KUKA KRL program: wkz4_off_st600.src, wkz4_off_st600.dat

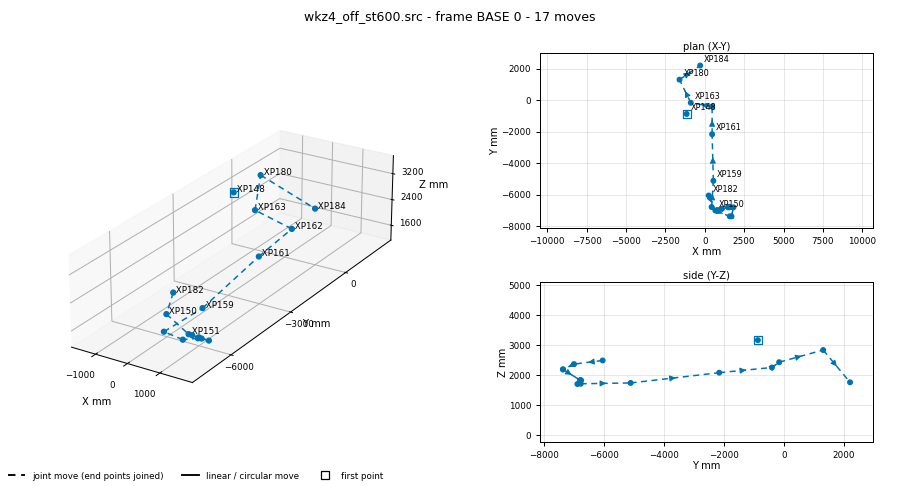
[picture p0: tool path of wkz4_off_st600.src in frame BASE 0, 17 of 18 moves have a stored position in this frame; points joined in program order, loops and branches not executed]
--- wkz4_off_st600.src ---
&ACCESS RVO1
&REL 256
&COMMENT Pega Griper ACCELO Geobox
&PARAM DISKPATH = KRC:\R1\Program
DEF wkz4_off_st600( )
;FOLD INI
  ;FOLD BASISTECH INI
    GLOBAL INTERRUPT DECL 3 WHEN $STOPMESS==TRUE DO IR_STOPM ( )
    INTERRUPT ON 3
    BAS (#INITMOV,0 )
  ;ENDFOLD (BASISTECH INI)
;FOLD GRIPPERTECH INI
USER_GRP(0,DUMMY,DUMMY,GDEFAULT)
;ENDFOLD (GRIPPERTECH INI)
  ;FOLD USER INI
    ;Make your modifications here

  ;ENDFOLD (USER INI)
;ENDFOLD (INI)

; Caracterização dos meios de produção:
; Versão Atual:
; 12/07/2013 12:00 Name: P13.050-R3 CHANGES: Pega Gripper na Geo
; Accelo

chk_w8_wechs_ok ( )       ; CHECK TOOLCHANGER

;FOLD PTP P148 CONT Vel=100 % PDAT114 Tool[4]:Gripper Lateral E.Accelo Base[0];%{PE}%R 8.2.20,%MKUKATPBASIS,%CMOVE,%VPTP,%P 1:PTP, 2:P148, 3:C_DIS, 5:100, 7:PDAT114
$BWDSTART=FALSE
PDAT_ACT=PPDAT114
FDAT_ACT=FP148
BAS(#PTP_PARAMS,100)
PTP XP148 C_DIS
;ENDFOLD
;FOLD PTP P172 CONT Vel=100 % PDAT131 Tool[4]:Gripper Lateral E.Accelo Base[0];%{PE}%R 8.2.20,%MKUKATPBASIS,%CMOVE,%VPTP,%P 1:PTP, 2:P172, 3:C_DIS, 5:100, 7:PDAT131
$BWDSTART=FALSE
PDAT_ACT=PPDAT131
FDAT_ACT=FP172
BAS(#PTP_PARAMS,100)
PTP XP172 C_DIS
;ENDFOLD
;FOLD PTP P182 Vel=100 % PDAT143 Tool[8]:Tool Changer Base[0];%{PE}%R 8.2.20,%MKUKATPBASIS,%CMOVE,%VPTP,%P 1:PTP, 2:P182, 3:, 5:100, 7:PDAT143
$BWDSTART=FALSE
PDAT_ACT=PPDAT143
FDAT_ACT=FP182
BAS(#PTP_PARAMS,100)
PTP XP182
;ENDFOLD


;FOLD OUT 3337 'R3 retira garra Geo' State=TRUE ;%{PE}%R 8.2.20,%MKUKATPBASIS,%COUT,%VOUTX,%P 2:3337, 3:R3 retira garra Geo, 5:TRUE, 6:
$OUT[3337]=TRUE
;ENDFOLD
;FOLD WAIT FOR ( IN 3337 'Aguarda Lib. entrar Geo' );%{PE}%R 8.2.20,%MKUKATPBASIS,%CEXT_WAIT_FOR,%VEXT_WAIT_FOR,%P 2:, 4:, 5:$IN, 6:3337, 7:Aguarda Lib. entrar Geo, 9:
WAIT FOR  ( $IN[3337] )
;ENDFOLD
;FOLD OUT 3337 'R3 retira garra Geo' State=FALSE ;%{PE}%R 8.2.20,%MKUKATPBASIS,%COUT,%VOUTX,%P 2:3337, 3:R3 retira garra Geo, 5:FALSE, 6:
$OUT[3337]=FALSE
;ENDFOLD
;FOLD OUT 3348 'Fora area GEOBOX' State=FALSE ;%{PE}%R 8.2.20,%MKUKATPBASIS,%COUT,%VOUTX,%P 2:3348, 3:Fora area GEOBOX, 5:FALSE, 6:
$OUT[3348]=FALSE
;ENDFOLD

;FOLD Collision.Monitoring_AREA_3_On ;%{PE}%MKUKATPUSER
COLLSTOP( 9, 1 ) ;not Interrupt-Controlled
;ENDFOLD
;FOLD Collision.Monitoring_AREA_5_On ;%{PE}%MKUKATPUSER
COLLSTOP( 11, 1 ) ;not Interrupt-Controlled
;ENDFOLD

;FOLD PTP P150 CONT Vel=100 % PDAT116 Tool[4]:Gripper Lateral E.Accelo Base[0];%{PE}%R 8.2.20,%MKUKATPBASIS,%CMOVE,%VPTP,%P 1:PTP, 2:P150, 3:C_DIS, 5:100, 7:PDAT116
$BWDSTART=FALSE
PDAT_ACT=PPDAT116
FDAT_ACT=FP150
BAS(#PTP_PARAMS,100)
PTP XP150 C_DIS
;ENDFOLD
;FOLD PTP P151 CONT Vel=100 % PDAT117 Tool[4]:Gripper Lateral E.Accelo Base[0];%{PE}%R 8.2.20,%MKUKATPBASIS,%CMOVE,%VPTP,%P 1:PTP, 2:P151, 3:C_DIS, 5:100, 7:PDAT117
$BWDSTART=FALSE
PDAT_ACT=PPDAT117
FDAT_ACT=FP151
BAS(#PTP_PARAMS,100)
PTP XP151 C_DIS
;ENDFOLD

;FOLD OUT 224 'Bloquear MPS' State=FALSE ;%{PE}%R 8.2.20,%MKUKATPBASIS,%COUT,%VOUTX,%P 2:224, 3:Bloquear MPS, 5:FALSE, 6:
$OUT[224]=FALSE
;ENDFOLD
;FOLD OUT 223 'Desbloquear MPS' State=TRUE ;%{PE}%R 8.2.20,%MKUKATPBASIS,%COUT,%VOUTX,%P 2:223, 3:Desbloquear MPS, 5:TRUE, 6:
$OUT[223]=TRUE
;ENDFOLD
;FOLD WAIT FOR ( IN 217 'MPS Destravado' );%{PE}%R 8.2.20,%MKUKATPBASIS,%CEXT_WAIT_FOR,%VEXT_WAIT_FOR,%P 2:, 4:, 5:$IN, 6:217, 7:MPS Destravado, 9:
WAIT FOR  ( $IN[217] )
;ENDFOLD
;FOLD WAIT FOR NOT ( IN 221 'MPS Travado' );%{PE}%R 8.2.20,%MKUKATPBASIS,%CEXT_WAIT_FOR,%VEXT_WAIT_FOR,%P 2:NOT, 4:, 5:$IN, 6:221, 7:MPS Travado, 9:
WAIT FOR  NOT ( $IN[221] )
;ENDFOLD

;FOLD ; PONTO DE PEGA DO GRIPPER;%{PE}%R 5.4.33,%MKUKATPBASIS,%CCOMMENT,%VNORMAL,%P 2:PONTO DE PEGA DO GRIPPER
;ENDFOLD
;FOLD LIN P179 Vel=2 m/s CPDAT55 Tool[8]:Tool Changer Base[0];%{PE}%R 8.2.20,%MKUKATPBASIS,%CMOVE,%VLIN,%P 1:LIN, 2:P179, 3:, 5:2, 7:CPDAT55
$BWDSTART=FALSE
LDAT_ACT=LCPDAT55
FDAT_ACT=FP179
BAS(#CP_PARAMS,2)
LIN XP179
;ENDFOLD

;FOLD WAIT Time=0.5 sec;%{PE}%R 8.2.20,%MKUKATPBASIS,%CWAIT,%VWAIT,%P 3:0.5
WAIT SEC 0.5
;ENDFOLD
;FOLD WAIT FOR ( IN 219 'Posicao p/ Acoplamento OK' );%{PE}%R 8.2.20,%MKUKATPBASIS,%CEXT_WAIT_FOR,%VEXT_WAIT_FOR,%P 2:, 4:, 5:$IN, 6:219, 7:Posicao p/ Acoplamento OK, 9:
WAIT FOR  ( $IN[219] )
;ENDFOLD
;FOLD OUT 223 'Desbloquear MPS' State=FALSE ;%{PE}%R 8.2.20,%MKUKATPBASIS,%COUT,%VOUTX,%P 2:223, 3:Desbloquear MPS, 5:FALSE, 6:
$OUT[223]=FALSE
;ENDFOLD
;FOLD OUT 224 'Bloquear MPS' State=TRUE ;%{PE}%R 8.2.20,%MKUKATPBASIS,%COUT,%VOUTX,%P 2:224, 3:Bloquear MPS, 5:TRUE, 6:
$OUT[224]=TRUE
;ENDFOLD
;FOLD WAIT FOR NOT ( IN 217 'MPS Destravado' );%{PE}%R 8.2.20,%MKUKATPBASIS,%CEXT_WAIT_FOR,%VEXT_WAIT_FOR,%P 2:NOT, 4:, 5:$IN, 6:217, 7:MPS Destravado, 9:
WAIT FOR  NOT ( $IN[217] )
;ENDFOLD
;FOLD WAIT FOR ( IN 221 'MPS Travado' );%{PE}%R 8.2.20,%MKUKATPBASIS,%CEXT_WAIT_FOR,%VEXT_WAIT_FOR,%P 2:, 4:, 5:$IN, 6:221, 7:MPS Travado, 9:
WAIT FOR  ( $IN[221] )
;ENDFOLD
;FOLD IBUS ON SEGMENT_3;%{PE}%R 8.2.20,%MKUKATPBASIS,%CIBUS,%VMAP,%P 2:#ON, 3:3
$IBUS_ON=IBUS_SEGMENT[3]
$IBUS_OFF=0
;ENDFOLD
;FOLD WAIT Time=0.5 sec;%{PE}%R 8.2.20,%MKUKATPBASIS,%CWAIT,%VWAIT,%P 3:0.5
WAIT SEC 0.5
;ENDFOLD

;FOLD OUT 3336 'R3 posição aguardando retirar garra' State=TRUE ;%{PE}%R 8.2.20,%MKUKATPBASIS,%COUT,%VOUTX,%P 2:3336, 3:R3 posição aguardando retirar garra, 5:TRUE, 6:
$OUT[3336]=TRUE
;ENDFOLD
;FOLD WAIT FOR ( IN 3335 'Aguarda Lib. entrar Geo' );%{PE}%R 8.2.20,%MKUKATPBASIS,%CEXT_WAIT_FOR,%VEXT_WAIT_FOR,%P 2:, 4:, 5:$IN, 6:3335, 7:Aguarda Lib. entrar Geo, 9:
WAIT FOR  ( $IN[3335] )
;ENDFOLD
;FOLD OUT 3336 'R3 posição aguardando retirar garra' State=FALSE ;%{PE}%R 8.2.20,%MKUKATPBASIS,%COUT,%VOUTX,%P 2:3336, 3:R3 posição aguardando retirar garra, 5:FALSE, 6:
$OUT[3336]=FALSE
;ENDFOLD

;FOLD SET Z1 ACCELO State=OPN GDAT14;%{PE}%R 8.2.1,%MKUKATPGRP,%CGRP,%VGRP,%P 2:6, 4:1, 5:#NO, 6:GDAT14, 8:0, 10:0
H50(GRP,6,1,GGDAT14)
;ENDFOLD
;FOLD SET Z2 ACCELO State=OPN GDAT15;%{PE}%R 8.2.1,%MKUKATPGRP,%CGRP,%VGRP,%P 2:7, 4:1, 5:#NO, 6:GDAT15, 8:0, 10:0
H50(GRP,7,1,GGDAT15)
;ENDFOLD
;FOLD SET Z3 ACCELO State= GDAT16;%{PE}%R 8.2.1,%MKUKATPGRP,%CGRP,%VGRP,%P 2:8, 4:1, 5:#NO, 6:GDAT16, 8:0, 10:0
H50(GRP,8,1,GGDAT16)
;ENDFOLD
;FOLD SET Z4 GRP Acello Bolha State=OPN GDAT18;%{PE}%R 8.2.1,%MKUKATPGRP,%CGRP,%VGRP,%P 2:16, 4:1, 5:#NO, 6:GDAT18, 8:0, 10:0
H50(GRP,16,1,GGDAT18)
;ENDFOLD
    chk_w4_grp1_opn()
    chk_w4_grp2_opn()
    chk_w4_grp3_opn()
    chk_w4_grp4_clo()

;FOLD LIN P155 CONT Vel=0.1 m/s CPDAT48 Tool[4]:Gripper Lateral E.Accelo Base[0];%{PE}%R 8.2.20,%MKUKATPBASIS,%CMOVE,%VLIN,%P 1:LIN, 2:P155, 3:C_DIS C_DIS, 5:0.1, 7:CPDAT48
$BWDSTART=FALSE
LDAT_ACT=LCPDAT48
FDAT_ACT=FP155
BAS(#CP_PARAMS,0.1)
LIN XP155 C_DIS C_DIS
;ENDFOLD

;FOLD PTP P170 CONT Vel=100 % PDAT140 Tool[4]:Gripper Lateral E.Accelo Base[0];%{PE}%R 8.2.20,%MKUKATPBASIS,%CMOVE,%VPTP,%P 1:PTP, 2:P170, 3:C_DIS, 5:100, 7:PDAT140
$BWDSTART=FALSE
PDAT_ACT=PPDAT140
FDAT_ACT=FP170
BAS(#PTP_PARAMS,100)
PTP XP170 C_DIS
;ENDFOLD
;FOLD PTP P181 CONT Vel=100 % PDAT139 Tool[4]:Gripper Lateral E.Accelo Base[0];%{PE}%R 8.2.20,%MKUKATPBASIS,%CMOVE,%VPTP,%P 1:PTP, 2:P181, 3:C_DIS, 5:100, 7:PDAT139
$BWDSTART=FALSE
PDAT_ACT=PPDAT139
FDAT_ACT=FP181
BAS(#PTP_PARAMS,100)
PTP XP181 C_DIS
;ENDFOLD

;FOLD WAIT FOR ( IN 219 'Posicao p/ Acoplamento OK' ) CONT;%{PE}%R 8.2.20,%MKUKATPBASIS,%CEXT_WAIT_FOR,%VEXT_WAIT_FOR,%P 2:, 4:, 5:$IN, 6:219, 7:Posicao p/ Acoplamento OK, 9:CONTINUE
CONTINUE
WAIT FOR  ( $IN[219] )
;ENDFOLD

;FOLD PTP P156 CONT Vel=100 % PDAT141 Tool[4]:Gripper Lateral E.Accelo Base[0];%{PE}%R 8.2.20,%MKUKATPBASIS,%CMOVE,%VPTP,%P 1:PTP, 2:P156, 3:C_DIS, 5:100, 7:PDAT141
$BWDSTART=FALSE
PDAT_ACT=PPDAT141
FDAT_ACT=FP156
BAS(#PTP_PARAMS,100)
PTP XP156 C_DIS
;ENDFOLD
;FOLD PTP P157 CONT Vel=100 % PDAT129 Tool[4]:Gripper Lateral E.Accelo Base[0];%{PE}%R 8.2.20,%MKUKATPBASIS,%CMOVE,%VPTP,%P 1:PTP, 2:P157, 3:C_DIS, 5:100, 7:PDAT129
$BWDSTART=FALSE
PDAT_ACT=PPDAT129
FDAT_ACT=FP157
BAS(#PTP_PARAMS,100)
PTP XP157 C_DIS
;ENDFOLD
;FOLD PTP P158 CONT Vel=100 % PDAT119 Tool[4]:Gripper Lateral E.Accelo Base[0];%{PE}%R 8.2.20,%MKUKATPBASIS,%CMOVE,%VPTP,%P 1:PTP, 2:P158, 3:C_DIS, 5:100, 7:PDAT119
$BWDSTART=FALSE
PDAT_ACT=PPDAT119
FDAT_ACT=FP158
BAS(#PTP_PARAMS,100)
PTP XP158 C_DIS
;ENDFOLD
;FOLD PTP P159 Vel=100 % PDAT120 Tool[4]:Gripper Lateral E.Accelo Base[0];%{PE}%R 8.2.20,%MKUKATPBASIS,%CMOVE,%VPTP,%P 1:PTP, 2:P159, 3:, 5:100, 7:PDAT120
$BWDSTART=FALSE
PDAT_ACT=PPDAT120
FDAT_ACT=FP159
BAS(#PTP_PARAMS,100)
PTP XP159
;ENDFOLD

;FOLD Collision.Monitoring_AREA_3_Off . ;%{PE}%MKUKATPUSER
COLLSTOP( 9, 2+0 )
;ENDFOLD
;FOLD Collision.Monitoring_AREA_5_Off . ;%{PE}%MKUKATPUSER
COLLSTOP( 11, 2+0 )
;ENDFOLD
;FOLD PULSE 3335 'R3 retirou garra da Geo' State=TRUE Time=3 sec;%{PE}%R 8.2.20,%MKUKATPBASIS,%COUT,%VPULSE,%P 2:3335, 3:R3 retirou garra da Geo, 5:TRUE, 6:, 8:3
PULSE($OUT[3335], TRUE,3)
;ENDFOLD
;FOLD OUT 3348 'Fora area GEOBOX' State=TRUE ;%{PE}%R 8.2.20,%MKUKATPBASIS,%COUT,%VOUTX,%P 2:3348, 3:Fora area GEOBOX, 5:TRUE, 6:
$OUT[3348]=TRUE
;ENDFOLD

start_weld_RESPOT()           ; Bit inicio solda respot

;FOLD PTP P161 CONT Vel=100 % PDAT122 Tool[4]:Gripper Lateral E.Accelo Base[0];%{PE}%R 8.2.20,%MKUKATPBASIS,%CMOVE,%VPTP,%P 1:PTP, 2:P161, 3:C_DIS, 5:100, 7:PDAT122
$BWDSTART=FALSE
PDAT_ACT=PPDAT122
FDAT_ACT=FP161
BAS(#PTP_PARAMS,100)
PTP XP161 C_DIS
;ENDFOLD
;FOLD PTP P162 CONT Vel=100 % PDAT123 Tool[4]:Gripper Lateral E.Accelo Base[0];%{PE}%R 8.2.20,%MKUKATPBASIS,%CMOVE,%VPTP,%P 1:PTP, 2:P162, 3:C_DIS, 5:100, 7:PDAT123
$BWDSTART=FALSE
PDAT_ACT=PPDAT123
FDAT_ACT=FP162
BAS(#PTP_PARAMS,100)
PTP XP162 C_DIS
;ENDFOLD
;FOLD PTP P163 CONT Vel=100 % PDAT124 Tool[4]:Gripper Lateral E.Accelo Base[0];%{PE}%R 8.2.20,%MKUKATPBASIS,%CMOVE,%VPTP,%P 1:PTP, 2:P163, 3:C_DIS, 5:100, 7:PDAT124
$BWDSTART=FALSE
PDAT_ACT=PPDAT124
FDAT_ACT=FP163
BAS(#PTP_PARAMS,100)
PTP XP163 C_DIS
;ENDFOLD
;FOLD PTP P180 CONT Vel=100 % PDAT138 Tool[4]:Gripper Lateral E.Accelo Base[0];%{PE}%R 8.2.20,%MKUKATPBASIS,%CMOVE,%VPTP,%P 1:PTP, 2:P180, 3:C_DIS, 5:100, 7:PDAT138
$BWDSTART=FALSE
PDAT_ACT=PPDAT138
FDAT_ACT=FP180
BAS(#PTP_PARAMS,100)
PTP XP180 C_DIS
;ENDFOLD
;FOLD PTP P184 Vel=100 % PDAT145 Tool[8]:Tool Changer Base[0];%{PE}%R 8.2.20,%MKUKATPBASIS,%CMOVE,%VPTP,%P 1:PTP, 2:P184, 3:, 5:100, 7:PDAT145
$BWDSTART=FALSE
PDAT_ACT=PPDAT145
FDAT_ACT=FP184
BAS(#PTP_PARAMS,100)
PTP XP184
;ENDFOLD

END

--- wkz4_off_st600.dat ---
&ACCESS RVO1
&REL 256
&COMMENT Pega Griper ACCELO Geobox
&PARAM DISKPATH = KRC:\R1\Program
DEFDAT  wkz4_off_st600
;FOLD EXTERNAL DECLARATIONS;%{PE}%MKUKATPBASIS,%CEXT,%VCOMMON,%P
;FOLD GRIPPERTECH EXT
EXT  H50 (INT  :IN,INT  :IN,INT  :IN,GRP_TYP  :IN )
;ENDFOLD (GRIPPERTECH EXT)
;FOLD SPOTTECH EXT

;ENDFOLD (SPOTTECH EXT)
;FOLD BASISTECH EXT;%{PE}%MKUKATPBASIS,%CEXT,%VEXT,%P
EXT  BAS (BAS_COMMAND  :IN,REAL  :IN )
DECL INT SUCCESS
;ENDFOLD (BASISTECH EXT)
;FOLD USER EXT;%{E}%MKUKATPUSER,%CEXT,%VEXT,%P
;Make your modifications here

;ENDFOLD (USER EXT)
;ENDFOLD (EXTERNAL DECLARATIONS)


;# ============ START PATH : bh_p13050r3_lta_01 =============
DECL BASIS_SUGG_T LAST_BASIS={POINT1[] "P1                      ",POINT2[] "P1                      ",CP_PARAMS[] "CPDAT0                  ",PTP_PARAMS[] "PDAT1                   ",CONT[] "                        ",CP_VEL[] "2.0                     ",PTP_VEL[] "100                     ",SYNC_PARAMS[] "SYNCDAT                 ",SPL_NAME[] "S0                      "}
DECL GRP_SUGG_T LAST_GRP={NUMBER[] "3                       ",STATE[] "1                       ",PARAMS[] "GDAT10                  "}
DECL GRP_TYP GGDAT2={G_APO #NO,GRP_TIME 0.200000003,CTRL #OFF,DLY 0,DST 1}
DECL GRP_TYP GGDAT7={G_APO #NO,GRP_TIME 0.200000003,CTRL #OFF,DLY 0,DST 1}
DECL GRP_TYP GGDAT8={G_APO #NO,GRP_TIME 0.200000003,CTRL #OFF,DLY 0,DST 1}
DECL GRP_TYP GGDAT9={G_APO #NO,GRP_TIME 0.200000003,CTRL #OFF,DLY 0,DST 1}
DECL GRP_TYP GGDAT10={G_APO #NO,GRP_TIME 0.200000003,CTRL #OFF,DLY 0,DST 1}
DECL PDAT PPDAT114={VEL 100.0,ACC 100.0,APO_DIST 100.0,APO_MODE #CDIS}
DECL E6POS XP148={X -1149.22803,Y -874.109619,Z 3176.2019,A 65.0211029,B 19.5584106,C -80.4266815,S 2,T 2,E1 1314.23999,E2 0.0,E3 0.0,E4 0.0,E5 0.0,E6 0.0}
DECL FDAT FP148={TOOL_NO 8,BASE_NO 0,IPO_FRAME #BASE,POINT2[] " ",TQ_STATE FALSE}
DECL PDAT PPDAT116={VEL 100.0,ACC 100.0,APO_DIST 100.0,APO_MODE #CDIS}
DECL E6POS XP150={X 672.64032,Y -7003.3418,Z 2375.8501,A -124.205002,B 65.71418,C -89.2604523,S 6,T 51,E1 5624.42578,E2 0.0,E3 0.0,E4 0.0,E5 0.0,E6 0.0}
DECL FDAT FP150={TOOL_NO 8,BASE_NO 0,IPO_FRAME #BASE,POINT2[] " ",TQ_STATE FALSE}
DECL PDAT PPDAT117={VEL 100.0,ACC 100.0,APO_DIST 100.0,APO_MODE #CDIS}
DECL E6POS XP151={X 1588.48303,Y -7373.36377,Z 2200.59106,A -90.2434692,B 75.2400208,C -90.1319809,S 6,T 51,E1 6474.80713,E2 0.0,E3 0.0,E4 0.0,E5 0.0,E6 0.0}
DECL FDAT FP151={TOOL_NO 8,BASE_NO 0,IPO_FRAME #BASE,POINT2[] " ",TQ_STATE FALSE}
DECL LDAT LCPDAT48={VEL 2.0,ACC 100.0,APO_DIST 100.0,APO_FAC 50.0,AXIS_VEL 100.0,AXIS_ACC 100.0,ORI_TYP #VAR,CIRC_TYP #BASE,JERK_FAC 50.0,GEAR_JERK 50.0,EXAX_IGN 0}
DECL E6POS XP155={X 1824.56006,Y -6798.22412,Z 1840.255,A 89.8839798,B -0.239819199,C 90.0336914,S 6,T 51,E1 6474.80811,E2 0.0,E3 0.0,E4 0.0,E5 0.0,E6 0.0}
DECL FDAT FP155={TOOL_NO 4,BASE_NO 0,IPO_FRAME #BASE,POINT2[] " ",TQ_STATE FALSE}
DECL E6POS XP156={X 1497.21301,Y -6805.64307,Z 1822.36902,A 79.8576965,B 0.419920802,C 92.5188293,S 6,T 51,E1 6307.34521,E2 0.0,E3 0.0,E4 0.0,E5 0.0,E6 0.0}
DECL FDAT FP156={TOOL_NO 4,BASE_NO 0,IPO_FRAME #BASE,POINT2[] " ",TQ_STATE FALSE}
DECL E6POS XP157={X 1091.43799,Y -6892.26807,Z 1713.03406,A 60.6017418,B 0.0325285792,C 102.3937,S 6,T 51,E1 5584.15283,E2 0.0,E3 0.0,E4 0.0,E5 0.0,E6 0.0}
DECL FDAT FP157={TOOL_NO 4,BASE_NO 0,IPO_FRAME #BASE,POINT2[] " ",TQ_STATE FALSE}
DECL PDAT PPDAT119={VEL 100.0,ACC 100.0,APO_DIST 100.0,APO_MODE #CDIS}
DECL E6POS XP158={X 435.602509,Y -6780.47119,Z 1722.00696,A 41.8793297,B -0.201007098,C 111.849503,S 6,T 51,E1 5011.26318,E2 0.0,E3 0.0,E4 0.0,E5 0.0,E6 0.0}
DECL FDAT FP158={TOOL_NO 4,BASE_NO 0,IPO_FRAME #BASE,POINT2[] " ",TQ_STATE FALSE}
DECL PDAT PPDAT120={VEL 100.0,ACC 100.0,APO_DIST 100.0,APO_MODE #CDIS}
DECL E6POS XP159={X 546.67218,Y -5117.54004,Z 1748.302,A 22.3437309,B -24.0161095,C 121.665398,S 6,T 51,E1 3181.00391,E2 0.0,E3 0.0,E4 0.0,E5 0.0,E6 0.0}
DECL FDAT FP159={TOOL_NO 4,BASE_NO 0,IPO_FRAME #BASE,POINT2[] " ",TQ_STATE FALSE}
DECL PDAT PPDAT122={VEL 100.0,ACC 100.0,APO_DIST 100.0,APO_MODE #CDIS}
DECL E6POS XP161={X 468.442993,Y -2162.86108,Z 2090.65503,A 55.5588303,B -37.0497398,C 119.3937,S 6,T 51,E1 957.071472,E2 0.0,E3 0.0,E4 0.0,E5 0.0,E6 0.0}
DECL FDAT FP161={TOOL_NO 4,BASE_NO 0,IPO_FRAME #BASE,POINT2[] " ",TQ_STATE FALSE}
DECL PDAT PPDAT123={VEL 100.0,ACC 100.0,APO_DIST 100.0,APO_MODE #CDIS}
DECL E6POS XP162={X 468.759094,Y -405.438202,Z 2263.58496,A 52.564209,B -8.07315445,C 107.346802,S 6,T 51,E1 -352.344513,E2 0.0,E3 0.0,E4 0.0,E5 0.0,E6 0.0}
DECL FDAT FP162={TOOL_NO 4,BASE_NO 0,IPO_FRAME #BASE,POINT2[] " ",TQ_STATE FALSE}
DECL PDAT PPDAT124={VEL 100.0,ACC 100.0,APO_DIST 100.0,APO_MODE #CDIS}
DECL E6POS XP163={X -886.202515,Y -164.792603,Z 2440.198,A -63.7987709,B 0.803352416,C 89.8370972,S 6,T 50,E1 -188.308807,E2 0.0,E3 0.0,E4 0.0,E5 0.0,E6 0.0}
DECL FDAT FP163={TOOL_NO 4,BASE_NO 0,IPO_FRAME #BASE,POINT2[] " ",TQ_STATE FALSE}
DECL GRP_TYP GGDAT11={G_APO #NO,GRP_TIME 0.200000003,CTRL #OFF,DLY 0,DST 1}
DECL GRP_TYP GGDAT12={G_APO #NO,GRP_TIME 0.200000003,CTRL #OFF,DLY 0,DST 1}
DECL GRP_TYP GGDAT13={G_APO #NO,GRP_TIME 0.200000003,CTRL #OFF,DLY 0,DST 1}
DECL E6POS XP170={X 1599.41296,Y -6791.38379,Z 1835.45996,A 89.5247116,B 0.314067394,C 90.0320206,S 6,T 51,E1 6508.55078,E2 0.0,E3 0.0,E4 0.0,E5 0.0,E6 0.0}
DECL FDAT FP170={TOOL_NO 4,BASE_NO 0,IPO_FRAME #BASE,POINT2[] " ",TQ_STATE FALSE}
DECL PDAT PPDAT129={VEL 100.0,ACC 100.0,APO_DIST 100.0,APO_MODE #CDIS}
DECL E6POS XP172={X -3332.60107,Y -3970.59692,Z 1629.59595,A -123.146202,B 34.176281,C 99.2101517,S 2,T 3,E1 1314.23999,E2 0.0,E3 0.0,E4 0.0,E5 0.0,E6 0.0}
DECL FDAT FP172={TOOL_NO 2,BASE_NO 2,IPO_FRAME #BASE,POINT2[] " ",TQ_STATE FALSE}
DECL PDAT PPDAT131={VEL 100.0,ACC 100.0,APO_DIST 100.0,APO_MODE #CDIS}
DECL E6POS XP179={X 1696.37305,Y -7373.36523,Z 2199.32495,A -90.2439423,B 75.2399902,C -90.1322708,S 6,T 51,E1 6474.80713,E2 0.0,E3 0.0,E4 0.0,E5 0.0,E6 0.0}
DECL FDAT FP179={TOOL_NO 8,BASE_NO 0,IPO_FRAME #BASE,POINT2[] " ",TQ_STATE FALSE}
DECL PDAT PPDAT138={VEL 100.0,ACC 100.0,APO_DIST 200.0,APO_MODE #CDIS}
DECL E6POS XP180={X -1601.43201,Y 1302.38696,Z 2846.13696,A -134.980698,B -60.753891,C 96.4850769,S 6,T 50,E1 -188.308395,E2 0.0,E3 0.0,E4 0.0,E5 0.0,E6 0.0}
DECL FDAT FP180={TOOL_NO 4,BASE_NO 0,IPO_FRAME #BASE,POINT2[] " ",TQ_STATE FALSE}
DECL E6POS XP181={X 1501.01404,Y -6769.40479,Z 1835.45496,A 89.5247421,B 0.314175397,C 90.0322189,S 6,T 51,E1 6508.55078,E2 0.0,E3 0.0,E4 0.0,E5 0.0,E6 0.0}
DECL FDAT FP181={TOOL_NO 4,BASE_NO 0,IPO_FRAME #BASE,POINT2[] " ",TQ_STATE FALSE}
DECL PDAT PPDAT139={VEL 100.0,ACC 100.0,APO_DIST 100.0,APO_MODE #CDIS}
DECL PDAT PPDAT140={VEL 100.0,ACC 100.0,APO_DIST 100.0,APO_MODE #CDIS}
DECL PDAT PPDAT141={VEL 100.0,ACC 100.0,APO_DIST 100.0,APO_MODE #CDIS}
DECL GRP_TYP GGDAT14={G_APO #NO,GRP_TIME 0.200000003,CTRL #OFF,DLY 0,DST 1}
DECL GRP_TYP GGDAT15={G_APO #NO,GRP_TIME 0.200000003,CTRL #OFF,DLY 0,DST 1}
DECL GRP_TYP GGDAT16={G_APO #NO,GRP_TIME 0.200000003,CTRL #OFF,DLY 0,DST 1}
DECL LDAT LCPDAT55={VEL 2.0,ACC 100.0,APO_DIST 100.0,APO_FAC 50.0,AXIS_VEL 100.0,AXIS_ACC 100.0,ORI_TYP #VAR,CIRC_TYP #BASE,JERK_FAC 50.0,GEAR_JERK 50.0,EXAX_IGN 0}
DECL E6POS XP182={X 251.264206,Y -6050.20996,Z 2498.62305,A -146.888901,B 53.0201111,C -84.5658264,S 6,T 51,E1 4487.74512,E2 0.0,E3 0.0,E4 0.0,E5 0.0,E6 0.0}
DECL FDAT FP182={TOOL_NO 8,BASE_NO 0,IPO_FRAME #BASE,POINT2[] " ",TQ_STATE FALSE}
DECL PDAT PPDAT143={VEL 100.0,ACC 100.0,APO_DIST 100.0,APO_MODE #CDIS}
DECL E6POS XP184={X -289.78421,Y 2198.16309,Z 1770.25806,A -171.851303,B 10.9435396,C 132.914993,S 2,T 34,E1 -188.312897,E2 0.0,E3 0.0,E4 0.0,E5 0.0,E6 0.0}
DECL FDAT FP184={TOOL_NO 8,BASE_NO 0,IPO_FRAME #BASE,POINT2[] " ",TQ_STATE FALSE}
DECL PDAT PPDAT145={VEL 100.0,ACC 100.0,APO_DIST 100.0}
DECL GRP_TYP GGDAT17={G_APO #NO,GRP_TIME 0.200000003,CTRL #OFF,DLY 0,DST 1}
DECL GRP_TYP GGDAT18={G_APO #NO,GRP_TIME 0.200000003,CTRL #OFF,DLY 0,DST 1}
DECL E6POS XP1={X 1107.651,Y 159.980301,Z 638.338013,A 0.305120289,B -89.7681503,C 89.5355377,S 6,T 51,E1 6474.81299,E2 0.0,E3 0.0,E4 0.0,E5 0.0,E6 0.0}
DECL FDAT FP1={TOOL_NO 5,BASE_NO 3,IPO_FRAME #BASE,POINT2[] " ",TQ_STATE FALSE}
DECL PDAT PPDAT1={VEL 100.0,ACC 100.0,APO_DIST 100.0}
ENDDAT
